PROGRAM Vision
VAR
END_VAR

//cyclic call to the vision operations
//seperate program assigned to seperate task and run on independant core of IPC
GVL_Vision.ImageChannel.CyclicLogic();

END_PROGRAM

(* stored: Version 1.1.0.1
   POU Vision: Id {df83cc56-7fa0-4916-abb7-796a92b5abde}, SpecialFunc None *)
